	    "T_FECHO_EV4.1_HMI".TON(IN := NOT "EV4.1",                  //Quando EV4.1 recebe sinal para fechar, inicia uma contagem
	                            PT := "Inputs_HMI".T_POS_EVS);
	                                                                //No final da contagem avalia se a EV está na posição pretendida
	                                                                
	    IF ("T_ABERTURA_EV4.1_HMI".Q AND (NOT "EV4.1_ABERTA" OR ("EV4.1_ABERTA" AND "EV4.1_FECHADA"))) OR   //Condição de avaria
	        ("T_FECHO_EV4.1_HMI".Q AND (NOT "EV4.1_FECHADA" OR ("EV4.1_ABERTA" AND "EV4.1_FECHADA"))) THEN
	        #"avaria_ev4.1" := TRUE;
	    ELSE
	        #"avaria_ev4.1" := FALSE;
	    END_IF;
	                                                                
	    IF #"avaria_ev4.1" = FALSE AND "EV4.1_ABERTA" AND NOT "EV4.1_FECHADA" THEN //Condição de EV4.1 ABERTA
	        "Estados_HMI"."EV4.1_ESTADO" := 1;
	        "Estados_HMI"."EV4.1_ESTADO_PAGCMD" := 1;
	    END_IF;
	    
	    
	    IF #"avaria_ev4.1" = FALSE AND "EV4.1_FECHADA" AND NOT "EV4.1_ABERTA" THEN //Condição de EV4.1 Fechada
	        "Estados_HMI"."EV4.1_ESTADO" := 0;
	        "Estados_HMI"."EV4.1_ESTADO_PAGCMD" := 0;
	    END_IF;
	    
	    
	    IF ("T_ABERTURA_EV4.1_HMI".Q AND (NOT "EV4.1_ABERTA" OR ("EV4.1_ABERTA" AND "EV4.1_FECHADA"))) OR   //Condição de avaria
	        ("T_FECHO_EV4.1_HMI".Q AND (NOT "EV4.1_FECHADA" OR ("EV4.1_ABERTA" AND "EV4.1_FECHADA"))) THEN
	        
	        "Estados_HMI"."EV4.1_ESTADO_PAGCMD" := 2;
	        
	        CASE #"temp_clock_0.625Hz" OF
	            0:
	                "Estados_HMI"."EV4.1_ESTADO" := 0;
	            1:
	                "Estados_HMI"."EV4.1_ESTADO" := 2;
	        END_CASE;
	    END_IF;
	    
	    IF "T_ABERTURA_EV4.1_HMI".Q = FALSE AND "T_FECHO_EV4.1_HMI".Q = FALSE AND
	        "EV4.1_ABERTA" = FALSE AND "EV4.1_FECHADA" = FALSE THEN  //Condição de transição das EVs
	        
	        "Estados_HMI"."EV4.1_ESTADO_PAGCMD" := 3;
	        
	        CASE #"temp_clock_0.625Hz" OF
	            0:
	                "Estados_HMI"."EV4.1_ESTADO" := 0;
	            1:
	                "Estados_HMI"."EV4.1_ESTADO" := 3;
	        END_CASE;
	    END_IF;
	    
	END_REGION
	
	REGION Estado_EV5.1
	    
	    "T_ABERTURA_EV5.1_HMI".TON(IN := "EV5.1",                   //Quando EV5.1 recebe sinal para abrir, inicia uma contagem
	                               PT := "Inputs_HMI".T_POS_EVS);
	    
	    "T_FECHO_EV5.1_HMI".TON(IN := NOT "EV5.1",                  //Quando EV5.1 recebe sinal para fechar, inicia uma contagem
	                            PT := "Inputs_HMI".T_POS_EVS);
	                                                                //No final da contagem avalia se a EV está na posição pretendida
	                                                                
	    IF ("T_ABERTURA_EV5.1_HMI".Q AND (NOT "EV5.1_ABERTA" OR ("EV5.1_ABERTA" AND "EV5.1_FECHADA"))) OR   //Condição de avaria
	        ("T_FECHO_EV5.1_HMI".Q AND (NOT "EV5.1_FECHADA" OR ("EV5.1_ABERTA" AND "EV5.1_FECHADA"))) THEN
	        #"avaria_ev5.1" := TRUE;
	    ELSE
	        #"avaria_ev5.1" := FALSE;
	    END_IF;
	                                                                
	    IF #"avaria_ev5.1" = FALSE AND "EV5.1_ABERTA" AND NOT "EV5.1_FECHADA" THEN //Condição de EV5.1 ABERTA
	        "Estados_HMI"."EV5.1_ESTADO" := 1;
	        "Estados_HMI"."EV5.1_ESTADO_PAGCMD" := 1;
	    END_IF;
	    
	    
	    IF #"avaria_ev5.1" = FALSE AND "EV5.1_FECHADA" AND NOT "EV5.1_ABERTA" THEN //Condição de EV5.1 Fechada
	        "Estados_HMI"."EV5.1_ESTADO" := 0;
	        "Estados_HMI"."EV5.1_ESTADO_PAGCMD" := 0;
	    END_IF;
	    
	    
	    IF ("T_ABERTURA_EV5.1_HMI".Q AND (NOT "EV5.1_ABERTA" OR ("EV5.1_ABERTA" AND "EV5.1_FECHADA"))) OR   //Condição de avaria
	        ("T_FECHO_EV5.1_HMI".Q AND (NOT "EV5.1_FECHADA" OR ("EV5.1_ABERTA" AND "EV5.1_FECHADA"))) THEN
	        
	        "Estados_HMI"."EV5.1_ESTADO_PAGCMD" := 2;
	        
	        CASE #"temp_clock_0.625Hz" OF
	            0:
	                "Estados_HMI"."EV5.1_ESTADO" := 0;
	            1:
	                "Estados_HMI"."EV5.1_ESTADO" := 2;
	        END_CASE;
	    END_IF;
	    
	    IF "T_ABERTURA_EV5.1_HMI".Q = FALSE AND "T_FECHO_EV5.1_HMI".Q = FALSE AND
	        "EV5.1_ABERTA" = FALSE AND "EV5.1_FECHADA" = FALSE THEN  //Condição de transição das EVs
	        
	        "Estados_HMI"."EV5.1_ESTADO_PAGCMD" := 3;
	        
	        CASE #"temp_clock_0.625Hz" OF
	            0:
	                "Estados_HMI"."EV5.1_ESTADO" := 0;
	            1:
	                "Estados_HMI"."EV5.1_ESTADO" := 3;
	        END_CASE;
	    END_IF;
	    
	END_REGION
	
	//FILTRO 2
	
	REGION Estado_EV1.2
	    "T_ABERTURA_EV1.2_HMI".TON(IN := "EV1.2",                   //Quando EV1.2 recebe sinal para abrir, inicia uma contagem
	                               PT := "Inputs_HMI".T_POS_EVS);
	    
	    "T_FECHO_EV1.2_HMI".TON(IN := NOT "EV1.2",                  //Quando EV1.2 recebe sinal para fechar, inicia uma contagem
	                            PT := "Inputs_HMI".T_POS_EVS);
	    //No final da contagem avalia se a EV está na posição pretendida
	    
	    IF ("T_ABERTURA_EV1.2_HMI".Q AND (NOT "EV1.2_ABERTA" OR ("EV1.2_ABERTA" AND "EV1.2_FECHADA"))) OR   //Condição de avaria
	        ("T_FECHO_EV1.2_HMI".Q AND (NOT "EV1.2_FECHADA" OR ("EV1.2_ABERTA" AND "EV1.2_FECHADA"))) THEN
	        #"avaria_ev1.2" := TRUE;
	    ELSE
	        #"avaria_ev1.2" := FALSE;
	    END_IF;
	        
	    IF #"avaria_ev1.2" = FALSE AND "EV1.2_ABERTA" AND NOT "EV1.2_FECHADA" THEN //Condição de EV1.2 ABERTA
	        "Estados_HMI"."EV1.2_ESTADO" := 1;
	        "Estados_HMI"."EV1.2_ESTADO_PAGCMD" := 1;
	    END_IF;
	    
	    
	    IF #"avaria_ev1.2" = FALSE AND "EV1.2_FECHADA" AND NOT "EV1.2_ABERTA" THEN //Condição de EV1.2 Fechada
	        "Estados_HMI"."EV1.2_ESTADO" := 0;
	        "Estados_HMI"."EV1.2_ESTADO_PAGCMD" := 0;
	    END_IF;
	    
	    
	    IF ("T_ABERTURA_EV1.2_HMI".Q AND (NOT "EV1.2_ABERTA" OR ("EV1.2_ABERTA" AND "EV1.2_FECHADA"))) OR   //Condição de avaria
	        ("T_FECHO_EV1.2_HMI".Q AND (NOT "EV1.2_FECHADA" OR ("EV1.2_ABERTA" AND "EV1.2_FECHADA"))) THEN
	        
	        "Estados_HMI"."EV1.2_ESTADO_PAGCMD" := 2;
	        
	        CASE #"temp_clock_0.625Hz" OF
	            0:
	                "Estados_HMI"."EV1.2_ESTADO" := 0;
	            1:
	                "Estados_HMI"."EV1.2_ESTADO" := 2;
	        END_CASE;
	    END_IF;
	    
	    IF "T_ABERTURA_EV1.2_HMI".Q = FALSE AND "T_FECHO_EV1.2_HMI".Q = FALSE AND
	        "EV1.2_ABERTA" = FALSE AND "EV1.2_FECHADA" = FALSE THEN  //Condição de transição das EVs
	        
	        "Estados_HMI"."EV1.2_ESTADO_PAGCMD" := 3;
	        
	        CASE #"temp_clock_0.625Hz" OF
	            0:
	                "Estados_HMI"."EV1.2_ESTADO" := 0;
	            1:
	                "Estados_HMI"."EV1.2_ESTADO" := 3;
	        END_CASE;
	    END_IF;
	    
	END_REGION
	
	REGION Estado_EV2.2
	    
	    "T_ABERTURA_EV2.2_HMI".TON(IN := "EV2.2",                   //Quando EV2.2 recebe sinal para abrir, inicia uma contagem
	                               PT := "Inputs_HMI".T_POS_EVS);
	    
	    "T_FECHO_EV2.2_HMI".TON(IN := NOT "EV2.2",                  //Quando EV2.2 recebe sinal para fechar, inicia uma contagem
	                            PT := "Inputs_HMI".T_POS_EVS);
	    //No final da contagem avalia se a EV está na posição pretendida
	    
	    IF ("T_ABERTURA_EV2.2_HMI".Q AND (NOT "EV2.2_ABERTA" OR ("EV2.2_ABERTA" AND "EV2.2_FECHADA"))) OR   //Condição de avaria
	        ("T_FECHO_EV2.2_HMI".Q AND (NOT "EV2.2_FECHADA" OR ("EV2.2_ABERTA" AND "EV2.2_FECHADA"))) THEN
	        #"avaria_ev2.2" := TRUE;
	    ELSE
	        #"avaria_ev2.2" := FALSE;
	    END_IF;
	    
	    IF #"avaria_ev2.2" = FALSE AND "EV2.2_ABERTA" AND NOT "EV2.2_FECHADA" THEN //Condição de EV2.2 ABERTA
	        "Estados_HMI"."EV2.2_ESTADO" := 1;
	        "Estados_HMI"."EV2.2_ESTADO_PAGCMD" := 1;
	    END_IF;
	    
	    
	    IF #"avaria_ev2.2" = FALSE AND "EV2.2_FECHADA" AND NOT "EV2.2_ABERTA" THEN //Condição de EV2.2 Fechada
	        "Estados_HMI"."EV2.2_ESTADO" := 0;
	        "Estados_HMI"."EV2.2_ESTADO_PAGCMD" := 0;
	    END_IF;
	    
	    
	    IF ("T_ABERTURA_EV2.2_HMI".Q AND (NOT "EV2.2_ABERTA" OR ("EV2.2_ABERTA" AND "EV2.2_FECHADA"))) OR   //Condição de avaria
	        ("T_FECHO_EV2.2_HMI".Q AND (NOT "EV2.2_FECHADA" OR ("EV2.2_ABERTA" AND "EV2.2_FECHADA"))) THEN
	        
	        "Estados_HMI"."EV2.2_ESTADO_PAGCMD" := 2;
	        
	        CASE #"temp_clock_0.625Hz" OF
	            0:
	                "Estados_HMI"."EV2.2_ESTADO" := 0;
	            1:
	                "Estados_HMI"."EV2.2_ESTADO" := 2;
	        END_CASE;
	    END_IF;
	    
	    IF "T_ABERTURA_EV2.2_HMI".Q = FALSE AND "T_FECHO_EV2.2_HMI".Q = FALSE AND
	        "EV2.2_ABERTA" = FALSE AND "EV2.2_FECHADA" = FALSE THEN  //Condição de transição das EVs
	        
	        "Estados_HMI"."EV2.2_ESTADO_PAGCMD" := 3;
	        
	        CASE #"temp_clock_0.625Hz" OF
	            0:
	                "Estados_HMI"."EV2.2_ESTADO" := 0;
	            1:
	                "Estados_HMI"."EV2.2_ESTADO" := 3;
	        END_CASE;
	    END_IF;
	    
	END_REGION
	
	REGION Estado_EV3.2
	    
	    "T_ABERTURA_EV3.2_HMI".TON(IN := "EV3.2",                   //Quando EV3.2 recebe sinal para abrir, inicia uma contagem
	                               PT := "Inputs_HMI".T_POS_EVS);
	    
	    "T_FECHO_EV3.2_HMI".TON(IN := NOT "EV3.2",                  //Quando EV3.2 recebe sinal para fechar, inicia uma contagem
	                            PT := "Inputs_HMI".T_POS_EVS);
	    //No final da contagem avalia se a EV está na posição pretendida
	    
	    IF ("T_ABERTURA_EV3.2_HMI".Q AND (NOT "EV3.2_ABERTA" OR ("EV3.2_ABERTA" AND "EV3.2_FECHADA"))) OR   //Condição de avaria
	        ("T_FECHO_EV3.2_HMI".Q AND (NOT "EV3.2_FECHADA" OR ("EV3.2_ABERTA" AND "EV3.2_FECHADA"))) THEN
	        #"avaria_ev3.2" := TRUE;
	    ELSE
	        #"avaria_ev3.2" := FALSE;
	    END_IF;
	        
	    
	    IF #"avaria_ev3.2" = FALSE AND "EV3.2_ABERTA" AND NOT "EV3.2_FECHADA" THEN //Condição de EV3.2 ABERTA
	        "Estados_HMI"."EV3.2_ESTADO" := 1;
	        "Estados_HMI"."EV3.2_ESTADO_PAGCMD" := 1;
	    END_IF;
	    
	    
	    IF #"avaria_ev3.2" = FALSE AND "EV3.2_FECHADA" AND NOT "EV3.2_ABERTA" THEN //Condição de EV3.2 Fechada
	        "Estados_HMI"."EV3.2_ESTADO" := 0;
	        "Estados_HMI"."EV3.2_ESTADO_PAGCMD" := 0;
	    END_IF;
	    
	    
	    IF ("T_ABERTURA_EV3.2_HMI".Q AND (NOT "EV3.2_ABERTA" OR ("EV3.2_ABERTA" AND "EV3.2_FECHADA"))) OR   //Condição de avaria
	        ("T_FECHO_EV3.2_HMI".Q AND (NOT "EV3.2_FECHADA" OR ("EV3.2_ABERTA" AND "EV3.2_FECHADA"))) THEN
	        
	        "Estados_HMI"."EV3.2_ESTADO_PAGCMD" := 2;
	        
	        CASE #"temp_clock_0.625Hz" OF
	            0:
	                "Estados_HMI"."EV3.2_ESTADO" := 0;
	            1:
	                "Estados_HMI"."EV3.2_ESTADO" := 2;
	        END_CASE;
	    END_IF;
	    
	    IF "T_ABERTURA_EV3.2_HMI".Q = FALSE AND "T_FECHO_EV3.2_HMI".Q = FALSE AND
	        "EV3.2_ABERTA" = FALSE AND "EV3.2_FECHADA" = FALSE THEN  //Condição de transição das EVs
	        
	        "Estados_HMI"."EV3.2_ESTADO_PAGCMD" := 3;
	        
	        CASE #"temp_clock_0.625Hz" OF
	            0:
	                "Estados_HMI"."EV3.2_ESTADO" := 0;
	            1:
	                "Estados_HMI"."EV3.2_ESTADO" := 3;
	        END_CASE;
	    END_IF;
	    
	END_REGION
	
	REGION Estado_EV4.2
	    
	    "T_ABERTURA_EV4.2_HMI".TON(IN := "EV4.2",                   //Quando EV4.2 recebe sinal para abrir, inicia uma contagem
	                               PT := "Inputs_HMI".T_POS_EVS);
	    
	    "T_FECHO_EV4.2_HMI".TON(IN := NOT "EV4.2",                  //Quando EV4.2 recebe sinal para fechar, inicia uma contagem
	                            PT := "Inputs_HMI".T_POS_EVS);
	    //No final da contagem avalia se a EV está na posição pretendida
	    
	    IF ("T_ABERTURA_EV4.2_HMI".Q AND (NOT "EV4.2_ABERTA" OR ("EV4.2_ABERTA" AND "EV4.2_FECHADA"))) OR   //Condição de avaria
	        ("T_FECHO_EV4.2_HMI".Q AND (NOT "EV4.2_FECHADA" OR ("EV4.2_ABERTA" AND "EV4.2_FECHADA"))) THEN
	        #"avaria_ev4.2" := TRUE;
	    ELSE
	        #"avaria_ev4.2" := FALSE;
	    END_IF;
	    
	    
	    IF #"avaria_ev4.2" = FALSE AND "EV4.2_ABERTA" AND NOT "EV4.2_FECHADA" THEN //Condição de EV4.2 ABERTA
	        "Estados_HMI"."EV4.2_ESTADO" := 1;
	        "Estados_HMI"."EV4.2_ESTADO_PAGCMD" := 1;
	    END_IF;
	    
	    
	    IF #"avaria_ev4.2" = FALSE AND "EV4.2_FECHADA" AND NOT "EV4.2_ABERTA" THEN //Condição de EV4.2 Fechada
	        "Estados_HMI"."EV4.2_ESTADO" := 0;
	        "Estados_HMI"."EV4.2_ESTADO_PAGCMD" := 0;
	    END_IF;
	    
	    
	    IF ("T_ABERTURA_EV4.2_HMI".Q AND (NOT "EV4.2_ABERTA" OR ("EV4.2_ABERTA" AND "EV4.2_FECHADA"))) OR   //Condição de avaria
	        ("T_FECHO_EV4.2_HMI".Q AND (NOT "EV4.2_FECHADA" OR ("EV4.2_ABERTA" AND "EV4.2_FECHADA"))) THEN
	        
	        "Estados_HMI"."EV4.2_ESTADO_PAGCMD" := 2;
	        
	        CASE #"temp_clock_0.625Hz" OF
	            0:
	                "Estados_HMI"."EV4.2_ESTADO" := 0;
	            1:
	                "Estados_HMI"."EV4.2_ESTADO" := 2;
	        END_CASE;
	    END_IF;
	    
	    IF "T_ABERTURA_EV4.2_HMI".Q = FALSE AND "T_FECHO_EV4.2_HMI".Q = FALSE AND
	        "EV4.2_ABERTA" = FALSE AND "EV4.2_FECHADA" = FALSE THEN  //Condição de transição das EVs
	        
	        "Estados_HMI"."EV4.2_ESTADO_PAGCMD" := 3;
	        
	        CASE #"temp_clock_0.625Hz" OF
	            0:
	                "Estados_HMI"."EV4.2_ESTADO" := 0;
	            1:
	                "Estados_HMI"."EV4.2_ESTADO" := 3;
	        END_CASE;
	    END_IF;
	    
	END_REGION
	
	REGION Estado_EV5.2
	    
	    "T_ABERTURA_EV5.2_HMI".TON(IN := "EV5.2",                   //Quando EV5.2 recebe sinal para abrir, inicia uma contagem
	                               PT := "Inputs_HMI".T_POS_EVS);
	    
	    "T_FECHO_EV5.2_HMI".TON(IN := NOT "EV5.2",                  //Quando EV5.2 recebe sinal para fechar, inicia uma contagem
	                            PT := "Inputs_HMI".T_POS_EVS);
	    //No final da contagem avalia se a EV está na posição pretendida
	    
	    IF ("T_ABERTURA_EV5.2_HMI".Q AND (NOT "EV5.2_ABERTA" OR ("EV5.2_ABERTA" AND "EV5.2_FECHADA"))) OR   //Condição de avaria
	        ("T_FECHO_EV5.2_HMI".Q AND (NOT "EV5.2_FECHADA" OR ("EV5.2_ABERTA" AND "EV5.2_FECHADA"))) THEN
	        #"avaria_ev5.2" := TRUE;
	    ELSE
	        #"avaria_ev5.2" := FALSE;
	    END_IF;
	    
	    
	    IF #"avaria_ev5.2" = FALSE AND "EV5.2_ABERTA" AND NOT "EV5.2_FECHADA" THEN //Condição de EV5.2 ABERTA
	        "Estados_HMI"."EV5.2_ESTADO" := 1;
	        "Estados_HMI"."EV5.2_ESTADO_PAGCMD" := 1;
	    END_IF;
	    
	    
	    IF #"avaria_ev5.2" = FALSE AND "EV5.2_FECHADA" AND NOT "EV5.2_ABERTA" THEN //Condição de EV5.2 Fechada
	        "Estados_HMI"."EV5.2_ESTADO" := 0;
	        "Estados_HMI"."EV5.2_ESTADO_PAGCMD" := 0;
	    END_IF;
	    
	    
	    IF ("T_ABERTURA_EV5.2_HMI".Q AND (NOT "EV5.2_ABERTA" OR ("EV5.2_ABERTA" AND "EV5.2_FECHADA"))) OR   //Condição de avaria
	        ("T_FECHO_EV5.2_HMI".Q AND (NOT "EV5.2_FECHADA" OR ("EV5.2_ABERTA" AND "EV5.2_FECHADA"))) THEN
	        
	        "Estados_HMI"."EV5.2_ESTADO_PAGCMD" := 2;
	        
	        CASE #"temp_clock_0.625Hz" OF
	            0:
	                "Estados_HMI"."EV5.2_ESTADO" := 0;
	            1:
	                "Estados_HMI"."EV5.2_ESTADO" := 2;
	        END_CASE;
	    END_IF;
	    
	    IF "T_ABERTURA_EV5.2_HMI".Q = FALSE AND "T_FECHO_EV5.2_HMI".Q = FALSE AND
	        "EV5.2_ABERTA" = FALSE AND "EV5.2_FECHADA" = FALSE THEN  //Condição de transição das EVs
	        
	        "Estados_HMI"."EV5.2_ESTADO_PAGCMD" := 3;
	        
	        CASE #"temp_clock_0.625Hz" OF
	            0:
	                "Estados_HMI"."EV5.2_ESTADO" := 0;
	            1:
	                "Estados_HMI"."EV5.2_ESTADO" := 3;
	        END_CASE;
	    END_IF;
	    
	END_REGION
END_FUNCTION

FUNCTION "Controlo_Pressostatos" : Void   // FC8, LAD
TITLE = Ao fim de 30s indica que atingiu setpoint de pressão
{ S7_Optimized_Access := 'TRUE' }
VERSION : 0.1
// stored: AutoNumber true, IsIECCheckEnabled false, SetENOAutomatically false, UDAEnableTagReadback false
BEGIN

REGION Network 1: Pressostato Filtro 1
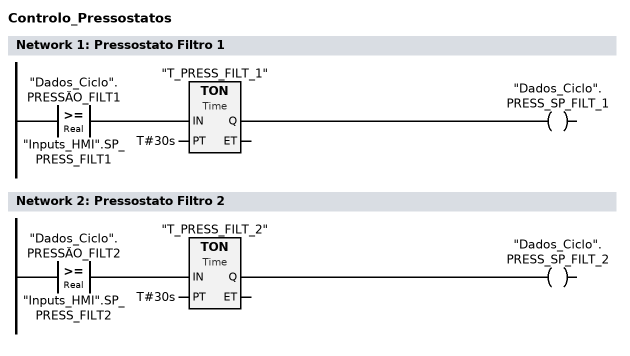
   RUNG wire#powerrail
      { S7_Templates := "SrcType := Real" } GE_Contact(in1 := "Dados_Ciclo".PRESSÃO_FILT1, in2 := "Inputs_HMI".SP_PRESS_FILT1)
      { S7_Templates := "time_type := Time" } "T_PRESS_FILT_1".TON(pt := T#30s, et =>)
      Coil( "Dados_Ciclo".PRESS_SP_FILT_1 )
   END_RUNG
   // the same network as SCL:
   "T_PRESS_FILT_1".TON(IN := "Dados_Ciclo".PRESSÃO_FILT1 >= "Inputs_HMI".SP_PRESS_FILT1, PT := T#30s);
   "Dados_Ciclo".PRESS_SP_FILT_1 := "T_PRESS_FILT_1".Q;
END_REGION

REGION Network 2: Pressostato Filtro 2
   RUNG wire#powerrail
      { S7_Templates := "SrcType := Real" } GE_Contact(in1 := "Dados_Ciclo".PRESSÃO_FILT2, in2 := "Inputs_HMI".SP_PRESS_FILT2)
      { S7_Templates := "time_type := Time" } "T_PRESS_FILT_2".TON(pt := T#30s, et =>)
      Coil( "Dados_Ciclo".PRESS_SP_FILT_2 )
   END_RUNG
   // the same network as SCL:
   "T_PRESS_FILT_2".TON(IN := "Dados_Ciclo".PRESSÃO_FILT2 >= "Inputs_HMI".SP_PRESS_FILT2, PT := T#30s);
   "Dados_Ciclo".PRESS_SP_FILT_2 := "T_PRESS_FILT_2".Q;
END_REGION
END_FUNCTION

FUNCTION "T_Func_Bombas" : Void   // FC9, LAD
{ S7_Optimized_Access := 'TRUE' }
VERSION : 0.1
// stored: AutoNumber true, IsIECCheckEnabled false, SetENOAutomatically false, UDAEnableTagReadback false
   VAR_TEMP   // added for the SCL form of the ladder/FBD networks
      _w1 : Bool;
   END_VAR
BEGIN

REGION Network 1: Período de tempo de alternancia das bombas
   // Se contador = 0, trabalha B1 e B2. Se = 1, trabalha B1 e B3. Se = 2, trabalha B2 e B3
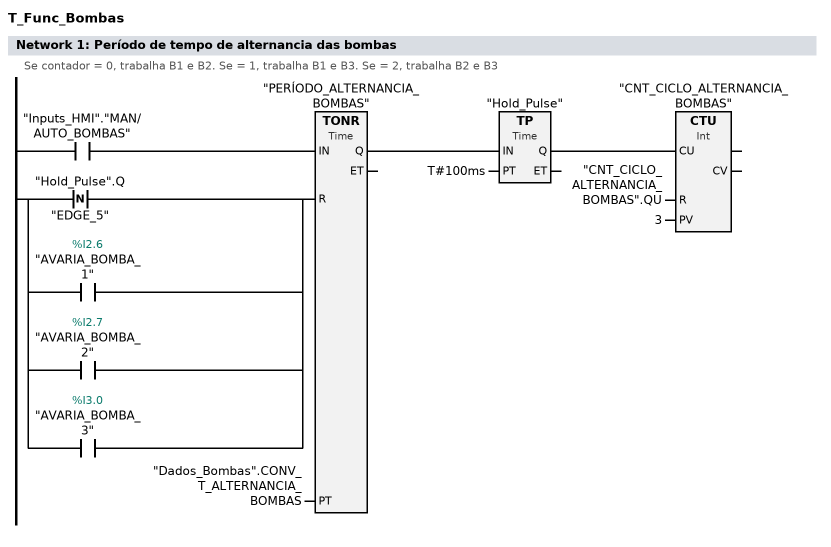
   RUNG wire#powerrail
      Contact( "Inputs_HMI"."MAN/AUTO_BOMBAS" )
      { S7_Templates := "time_type := Time" } "PERÍODO_ALTERNANCIA_BOMBAS".TONR(r := wire#w1, pt := "Dados_Bombas".CONV_T_ALTERNANCIA_BOMBAS, et =>)
      { S7_Templates := "time_type := Time" } "Hold_Pulse".TP(pt := T#100ms, et =>)
      { S7_Templates := "value_type := Int" } "CNT_CICLO_ALTERNANCIA_BOMBAS".CTU(r := "CNT_CICLO_ALTERNANCIA_BOMBAS".QU, pv := 3, cv =>)
   END_RUNG
   RUNG wire#powerrail
      N_Contact(operand := "Hold_Pulse".Q, bit := "EDGE_5")
   END_RUNG wire#w1
   RUNG wire#powerrail
      Contact( "AVARIA_BOMBA_1" )
   END_RUNG wire#w1
   RUNG wire#powerrail
      Contact( "AVARIA_BOMBA_2" )
   END_RUNG wire#w1
   RUNG wire#powerrail
      Contact( "AVARIA_BOMBA_3" )
   END_RUNG wire#w1
   // the same network as SCL:
   #_w1 := NOT "Hold_Pulse".Q AND "EDGE_5";   // falling edge of "Hold_Pulse".Q
   "EDGE_5" := "Hold_Pulse".Q;
   "PERÍODO_ALTERNANCIA_BOMBAS".TONR(IN := "Inputs_HMI"."MAN/AUTO_BOMBAS",
                           R := #_w1 OR "AVARIA_BOMBA_1" OR "AVARIA_BOMBA_2" OR "AVARIA_BOMBA_3",
                           PT := "Dados_Bombas".CONV_T_ALTERNANCIA_BOMBAS);
   "Hold_Pulse".TP(IN := "PERÍODO_ALTERNANCIA_BOMBAS".Q, PT := T#100ms);
   "CNT_CICLO_ALTERNANCIA_BOMBAS".CTU(CU := "Hold_Pulse".Q, R := "CNT_CICLO_ALTERNANCIA_BOMBAS".QU, PV := 3);
END_REGION
END_FUNCTION

FUNCTION "Conversão_Tempo_Bombas" : Void
{ S7_Optimized_Access := 'TRUE' }
VERSION : 0.1
   VAR_TEMP 
      decimal_b2 : Real;
      result_b2 : Real;
      decimal_b3 : Real;
      result_b3 : Real;
      decimal_TON : Real;
      decimal_TOFF : Real;
      result_TON : Real;
      result_TOFF : Real;
   END_VAR


BEGIN
	//Conversão do tempo de alternancia das bombas introduzido na hmi (ex: em vez de introduzir 1.5 para dar 1h30m,
	//introduz-se 1.3 para da 1h30m
	
	
	//conversão T_ALTERNANCIA bombas 
	//
	#decimal_TON := ("Inputs_HMI".T_ALTERNANCIA_BOMBAS - TRUNC("Inputs_HMI".T_ALTERNANCIA_BOMBAS)) * 1.6667;
	#result_TON := TRUNC("Inputs_HMI".T_ALTERNANCIA_BOMBAS) + #decimal_TON;
	
	"Dados_Bombas".CONV_T_ALTERNANCIA_BOMBAS :=
	DINT_TO_TIME(
	             REAL_TO_DINT(#result_TON * 3600000));
	
	
	REGION leitura_tempos_func_bombas_para_hmi
	    
	    
	    "Dados_Bombas".HORAS_TON_B1 := "CNT_FUNC_B1".CV;
	    
	    "Dados_Bombas".HORAS_TON_B2 := "CNT_FUNC_B2".CV;
	    
	    "Dados_Bombas".HORAS_TON_B3 := "CNT_FUNC_B3".CV;
	   
	END_REGION
	
END_FUNCTION

FUNCTION "Encrav_Inputs_HMI" : Void
{ S7_Optimized_Access := 'TRUE' }
VERSION : 0.1

BEGIN
	IF "Inputs_HMI"."MAN/AUTO_BOMBAS" = TRUE THEN
	    
	    "Inputs_HMI".ON_OFF_BOMBA_1 := FALSE;
	    "Inputs_HMI".ON_OFF_BOMBA_2 := FALSE;
	    "Inputs_HMI".ON_OFF_BOMBA_3 := FALSE;
	    
	END_IF;
	
	IF "Inputs_HMI"."MAN/AUTO" = TRUE THEN
	    
	    "Inputs_HMI"."ON_OFF_EV1.1" := FALSE;
	    "Inputs_HMI"."ON_OFF_EV2.1" := FALSE;
	    "Inputs_HMI"."ON_OFF_EV3.1" := FALSE;
	    "Inputs_HMI"."ON_OFF_EV4.1" := FALSE;
	    "Inputs_HMI"."ON_OFF_EV5.1" := FALSE;
	    
	    "Inputs_HMI"."ON_OFF_EV1.2" := FALSE;
	    "Inputs_HMI"."ON_OFF_EV2.2" := FALSE;
	    "Inputs_HMI"."ON_OFF_EV3.2" := FALSE;
	    "Inputs_HMI"."ON_OFF_EV4.2" := FALSE;
	    "Inputs_HMI"."ON_OFF_EV5.2" := FALSE;
	 
	END_IF;
	
END_FUNCTION

FUNCTION "Conversão_TLAV_TRINSE" : Void
{ S7_Optimized_Access := 'TRUE' }
VERSION : 0.1

BEGIN
	//Conversão do tempo decorrido de lavagem e enxaguamento para minutos
	
	"Estados_HMI".T_LAV_MINUTOS := (TIME_TO_DINT("T_LAVAGEM".ET) MOD 3600000) / 60000;
	"Estados_HMI".T_RINSE_MINUTOS := (TIME_TO_DINT("T_RINSE".ET) MOD 3600000) / 60000;
END_FUNCTION

FUNCTION "Alarmes" : Void
{ S7_Optimized_Access := 'TRUE' }
VERSION : 0.1

BEGIN
	//Alarmes filtro 1
	//
	REGION ALARME_V1.1
	    IF "T_ABERTURA_EV1.1_HMI".Q AND NOT "EV1.1_ABERTA" THEN  //Válvula não abriu
	        "Estados_HMI".ALARMES_LISTA_1.%X0 := TRUE;
	    ELSE
	        "Estados_HMI".ALARMES_LISTA_1.%X0 := FALSE;
	    END_IF;
	    
	    
	    IF "T_ABERTURA_EV1.1_HMI".Q AND "EV1.1_ABERTA" AND "EV1.1_FECHADA" THEN  //Avaria fim de curso de fecho
	        "Estados_HMI".ALARMES_LISTA_1.%X1 := TRUE;
	    ELSE
	        "Estados_HMI".ALARMES_LISTA_1.%X1 := FALSE;
	    END_IF;
	    
	    
	    IF "T_FECHO_EV1.1_HMI".Q AND NOT "EV1.1_FECHADA" THEN  //Válvula não fechou
	        "Estados_HMI".ALARMES_LISTA_1.%X2 := TRUE;
	    ELSE
	        "Estados_HMI".ALARMES_LISTA_1.%X2 := FALSE;
	    END_IF;
	    
	    
	    IF "T_FECHO_EV1.1_HMI".Q AND "EV1.1_ABERTA" AND "EV1.1_FECHADA" THEN  //Avaria fim de curso de abertura
	        "Estados_HMI".ALARMES_LISTA_1.%X3 := TRUE;
	    ELSE
	        "Estados_HMI".ALARMES_LISTA_1.%X3 := FALSE;
	    END_IF;
	END_REGION
	REGION ALARME_V2.1
	    IF "T_ABERTURA_EV2.1_HMI".Q AND NOT "EV2.1_ABERTA" THEN  //Válvula não abriu
	        "Estados_HMI".ALARMES_LISTA_1.%X4 := TRUE;
	    ELSE
	        "Estados_HMI".ALARMES_LISTA_1.%X4 := FALSE;
	    END_IF;
	    
	    
	    IF "T_ABERTURA_EV2.1_HMI".Q AND "EV2.1_ABERTA" AND "EV2.1_FECHADA" THEN  //Avaria fim de curso de fecho
	        "Estados_HMI".ALARMES_LISTA_1.%X5 := TRUE;
	    ELSE
	        "Estados_HMI".ALARMES_LISTA_1.%X5 := FALSE;
	    END_IF;
	    
	    
	    IF "T_FECHO_EV2.1_HMI".Q AND NOT "EV2.1_FECHADA" THEN  //Válvula não fechou
	        "Estados_HMI".ALARMES_LISTA_1.%X6 := TRUE;
	    ELSE
	        "Estados_HMI".ALARMES_LISTA_1.%X6 := FALSE;
	    END_IF;
	    
	    
	    IF "T_FECHO_EV2.1_HMI".Q AND "EV2.1_ABERTA" AND "EV2.1_FECHADA" THEN  //Avaria fim de curso de abertura
	        "Estados_HMI".ALARMES_LISTA_1.%X7 := TRUE;
	    ELSE
	        "Estados_HMI".ALARMES_LISTA_1.%X7 := FALSE;
	    END_IF;
	END_REGION
	REGION ALARME_V3.1
	    IF "T_ABERTURA_EV3.1_HMI".Q AND NOT "EV3.1_ABERTA" THEN  //Válvula não abriu
	        "Estados_HMI".ALARMES_LISTA_1.%X8 := TRUE;
	    ELSE
	        "Estados_HMI".ALARMES_LISTA_1.%X8 := FALSE;
	    END_IF;
	    
	    
	    IF "T_ABERTURA_EV3.1_HMI".Q AND "EV3.1_ABERTA" AND "EV3.1_FECHADA" THEN  //Avaria fim de curso de fecho
	        "Estados_HMI".ALARMES_LISTA_1.%X9 := TRUE;
	    ELSE
	        "Estados_HMI".ALARMES_LISTA_1.%X9 := FALSE;
	    END_IF;
	    
	    
	    IF "T_FECHO_EV3.1_HMI".Q AND NOT "EV3.1_FECHADA" THEN  //Válvula não fechou
	        "Estados_HMI".ALARMES_LISTA_1.%X10 := TRUE;
	    ELSE
	        "Estados_HMI".ALARMES_LISTA_1.%X10 := FALSE;
	    END_IF;
	    
	    
	    IF "T_FECHO_EV3.1_HMI".Q AND "EV3.1_ABERTA" AND "EV3.1_FECHADA" THEN  //Avaria fim de curso de abertura
	        "Estados_HMI".ALARMES_LISTA_1.%X11 := TRUE;
	    ELSE
	        "Estados_HMI".ALARMES_LISTA_1.%X11 := FALSE;
	    END_IF;
	END_REGION
	REGION ALARME_V4.1
	    IF "T_ABERTURA_EV4.1_HMI".Q AND NOT "EV4.1_ABERTA" THEN  //Válvula não abriu
	        "Estados_HMI".ALARMES_LISTA_1.%X12 := TRUE;
	    ELSE
	        "Estados_HMI".ALARMES_LISTA_1.%X12 := FALSE;
	    END_IF;
	    
	    
	    IF "T_ABERTURA_EV4.1_HMI".Q AND "EV4.1_ABERTA" AND "EV4.1_FECHADA" THEN  //Avaria fim de curso de fecho
	        "Estados_HMI".ALARMES_LISTA_1.%X13 := TRUE;
	    ELSE
	        "Estados_HMI".ALARMES_LISTA_1.%X13 := FALSE;
	    END_IF;
	    
	    
	    IF "T_FECHO_EV4.1_HMI".Q AND NOT "EV4.1_FECHADA" THEN  //Válvula não fechou
	        "Estados_HMI".ALARMES_LISTA_1.%X14 := TRUE;
	    ELSE
	        "Estados_HMI".ALARMES_LISTA_1.%X14 := FALSE;
	    END_IF;
	    
	    
	    IF "T_FECHO_EV4.1_HMI".Q AND "EV4.1_ABERTA" AND "EV4.1_FECHADA" THEN  //Avaria fim de curso de abertura
	        "Estados_HMI".ALARMES_LISTA_1.%X15 := TRUE;
	    ELSE
	        "Estados_HMI".ALARMES_LISTA_1.%X15 := FALSE;
	    END_IF;
	END_REGION
	REGION ALARME_V5.1
	    IF "T_ABERTURA_EV5.1_HMI".Q AND NOT "EV5.1_ABERTA" THEN  //Válvula não abriu
	        "Estados_HMI".ALARMES_LISTA_2.%X0 := TRUE;
	    ELSE
	        "Estados_HMI".ALARMES_LISTA_2.%X0 := FALSE;
	    END_IF;
	    
	    
	    IF "T_ABERTURA_EV5.1_HMI".Q AND "EV5.1_ABERTA" AND "EV5.1_FECHADA" THEN  //Avaria fim de curso de fecho
	        "Estados_HMI".ALARMES_LISTA_2.%X1 := TRUE;
	    ELSE
	        "Estados_HMI".ALARMES_LISTA_2.%X1 := FALSE;
	    END_IF;
	    
	    
	    IF "T_FECHO_EV5.1_HMI".Q AND NOT "EV5.1_FECHADA" THEN  //Válvula não fechou
	        "Estados_HMI".ALARMES_LISTA_2.%X2 := TRUE;
	    ELSE
	        "Estados_HMI".ALARMES_LISTA_2.%X2 := FALSE;
	    END_IF;
	    
	    
	    IF "T_FECHO_EV5.1_HMI".Q AND "EV5.1_ABERTA" AND "EV5.1_FECHADA" THEN  //Avaria fim de curso de abertura
	        "Estados_HMI".ALARMES_LISTA_2.%X3 := TRUE;
	    ELSE
	        "Estados_HMI".ALARMES_LISTA_2.%X3 := FALSE;
	    END_IF;
	END_REGION
	
	//Alarmes filtro 2
	//
	REGION ALARME_V1.2
	    IF "T_ABERTURA_EV1.2_HMI".Q AND NOT "EV1.2_ABERTA" THEN  //Válvula não abriu
	        "Estados_HMI".ALARMES_LISTA_2.%X4 := TRUE;
	    ELSE
	        "Estados_HMI".ALARMES_LISTA_2.%X4 := FALSE;
	    END_IF;
	    
	    
	    IF "T_ABERTURA_EV1.2_HMI".Q AND "EV1.2_ABERTA" AND "EV1.2_FECHADA" THEN  //Avaria fim de curso de fecho
	        "Estados_HMI".ALARMES_LISTA_2.%X5 := TRUE;
	    ELSE
	        "Estados_HMI".ALARMES_LISTA_2.%X5 := FALSE;
	    END_IF;
	    
	    
	    IF "T_FECHO_EV1.2_HMI".Q AND NOT "EV1.2_FECHADA" THEN  //Válvula não fechou
	        "Estados_HMI".ALARMES_LISTA_2.%X6 := TRUE;
	    ELSE
	        "Estados_HMI".ALARMES_LISTA_2.%X6 := FALSE;
	    END_IF;
	    
	    
	    IF "T_FECHO_EV1.2_HMI".Q AND "EV1.2_ABERTA" AND "EV1.2_FECHADA" THEN  //Avaria fim de curso de abertura
	        "Estados_HMI".ALARMES_LISTA_2.%X7 := TRUE;
	    ELSE
	        "Estados_HMI".ALARMES_LISTA_2.%X7 := FALSE;
	    END_IF;
	END_REGION
	REGION ALARME_V2.2
	    IF "T_ABERTURA_EV2.2_HMI".Q AND NOT "EV2.2_ABERTA" THEN  //Válvula não abriu
	        "Estados_HMI".ALARMES_LISTA_2.%X8 := TRUE;
	    ELSE
	        "Estados_HMI".ALARMES_LISTA_2.%X8 := FALSE;
	    END_IF;
	    
	    
	    IF "T_ABERTURA_EV2.2_HMI".Q AND "EV2.2_ABERTA" AND "EV2.2_FECHADA" THEN  //Avaria fim de curso de fecho
	        "Estados_HMI".ALARMES_LISTA_2.%X9 := TRUE;
	    ELSE
	        "Estados_HMI".ALARMES_LISTA_2.%X9 := FALSE;
	    END_IF;
	    
	    
	    IF "T_FECHO_EV2.2_HMI".Q AND NOT "EV2.2_FECHADA" THEN  //Válvula não fechou
	        "Estados_HMI".ALARMES_LISTA_2.%X10 := TRUE;
	    ELSE
	        "Estados_HMI".ALARMES_LISTA_2.%X10 := FALSE;
	    END_IF;
	    
	    
	    IF "T_FECHO_EV2.2_HMI".Q AND "EV2.2_ABERTA" AND "EV2.2_FECHADA" THEN  //Avaria fim de curso de abertura
	        "Estados_HMI".ALARMES_LISTA_2.%X11 := TRUE;
	    ELSE
	        "Estados_HMI".ALARMES_LISTA_2.%X11 := FALSE;
	    END_IF;
	END_REGION
	REGION ALARME_V3.2
	    IF "T_ABERTURA_EV3.2_HMI".Q AND NOT "EV3.2_ABERTA" THEN  //Válvula não abriu
	        "Estados_HMI".ALARMES_LISTA_2.%X12 := TRUE;
	    ELSE
	        "Estados_HMI".ALARMES_LISTA_2.%X12 := FALSE;
	    END_IF;
	    
	    
	    IF "T_ABERTURA_EV3.2_HMI".Q AND "EV3.2_ABERTA" AND "EV3.2_FECHADA" THEN  //Avaria fim de curso de fecho
	        "Estados_HMI".ALARMES_LISTA_2.%X13 := TRUE;
	    ELSE
	        "Estados_HMI".ALARMES_LISTA_2.%X13 := FALSE;
	    END_IF;
	    
	    
	    IF "T_FECHO_EV3.2_HMI".Q AND NOT "EV3.2_FECHADA" THEN  //Válvula não fechou
	        "Estados_HMI".ALARMES_LISTA_2.%X14 := TRUE;
	    ELSE
	        "Estados_HMI".ALARMES_LISTA_2.%X14 := FALSE;
	    END_IF;
	    
	    
	    IF "T_FECHO_EV3.2_HMI".Q AND "EV3.2_ABERTA" AND "EV3.2_FECHADA" THEN  //Avaria fim de curso de abertura
	        "Estados_HMI".ALARMES_LISTA_2.%X15 := TRUE;
	    ELSE
	        "Estados_HMI".ALARMES_LISTA_2.%X15 := FALSE;
	    END_IF;
	END_REGION
	REGION ALARME_V4.2
	    IF "T_ABERTURA_EV4.2_HMI".Q AND NOT "EV4.2_ABERTA" THEN  //Válvula não abriu
	        "Estados_HMI".ALARMES_LISTA_3.%X0 := TRUE;
	    ELSE
	        "Estados_HMI".ALARMES_LISTA_3.%X0 := FALSE;
	    END_IF;
	    
	    
	    IF "T_ABERTURA_EV4.2_HMI".Q AND "EV4.2_ABERTA" AND "EV4.2_FECHADA" THEN  //Avaria fim de curso de fecho
	        "Estados_HMI".ALARMES_LISTA_3.%X1 := TRUE;
	    ELSE
	        "Estados_HMI".ALARMES_LISTA_3.%X1 := FALSE;
	    END_IF;
	    
	    
	    IF "T_FECHO_EV4.2_HMI".Q AND NOT "EV4.2_FECHADA" THEN  //Válvula não fechou
	        "Estados_HMI".ALARMES_LISTA_3.%X2 := TRUE;
	    ELSE
	        "Estados_HMI".ALARMES_LISTA_3.%X2 := FALSE;
	    END_IF;
	    
	    
	    IF "T_FECHO_EV4.2_HMI".Q AND "EV4.2_ABERTA" AND "EV4.2_FECHADA" THEN  //Avaria fim de curso de abertura
	        "Estados_HMI".ALARMES_LISTA_3.%X3 := TRUE;
	    ELSE
	        "Estados_HMI".ALARMES_LISTA_3.%X3 := FALSE;
	    END_IF;
	END_REGION
	REGION ALARME_V5.2
	    IF "T_ABERTURA_EV5.2_HMI".Q AND NOT "EV5.2_ABERTA" THEN  //Válvula não abriu
	        "Estados_HMI".ALARMES_LISTA_3.%X4 := TRUE;
	    ELSE
	        "Estados_HMI".ALARMES_LISTA_3.%X4 := FALSE;
	    END_IF;
	    
	    
	    IF "T_ABERTURA_EV5.2_HMI".Q AND "EV5.2_ABERTA" AND "EV5.2_FECHADA" THEN  //Avaria fim de curso de fecho
	        "Estados_HMI".ALARMES_LISTA_3.%X5 := TRUE;
	    ELSE
	        "Estados_HMI".ALARMES_LISTA_3.%X5 := FALSE;
	    END_IF;
	    
	    
	    IF "T_FECHO_EV5.2_HMI".Q AND NOT "EV5.2_FECHADA" THEN  //Válvula não fechou
	        "Estados_HMI".ALARMES_LISTA_3.%X6 := TRUE;
	    ELSE
	        "Estados_HMI".ALARMES_LISTA_3.%X6 := FALSE;
	    END_IF;
	    
	    
	    IF "T_FECHO_EV5.2_HMI".Q AND "EV5.2_ABERTA" AND "EV5.2_FECHADA" THEN  //Avaria fim de curso de abertura
	        "Estados_HMI".ALARMES_LISTA_3.%X7 := TRUE;
	    ELSE
	        "Estados_HMI".ALARMES_LISTA_3.%X7 := FALSE;
	    END_IF;
	END_REGION
	
	//Alarmes Bombas
	//
	REGION ALARME_BOMBA_1
	    IF "AVARIA_BOMBA_1" = TRUE THEN
	        "Estados_HMI".ALARMES_LISTA_3.%X8 := TRUE;
	    ELSE
	        "Estados_HMI".ALARMES_LISTA_3.%X8 := FALSE;
	    END_IF;
	END_REGION
	
	REGION ALARME_BOMBA_2
	    IF "AVARIA_BOMBA_2" = TRUE THEN
	        "Estados_HMI".ALARMES_LISTA_3.%X9 := TRUE;
	    ELSE
	        "Estados_HMI".ALARMES_LISTA_3.%X9 := FALSE;
	    END_IF;
	END_REGION
	
	REGION ALARME_BOMBA_3
	    IF "AVARIA_BOMBA_3" = TRUE THEN
	        "Estados_HMI".ALARMES_LISTA_3.%X10 := TRUE;
	    ELSE
	        "Estados_HMI".ALARMES_LISTA_3.%X10 := FALSE;
	    END_IF;
	END_REGION
	
	
	
	
	
	
END_FUNCTION

FUNCTION "UV" : Void   // FC15, LAD
{ S7_Optimized_Access := 'TRUE' }
VERSION : 0.1
// stored: AutoNumber true, IsIECCheckEnabled false, SetENOAutomatically false, UDAEnableTagReadback false
   VAR_TEMP
      sr_ultravioleta : Bool;
   END_VAR
BEGIN

REGION Network 1
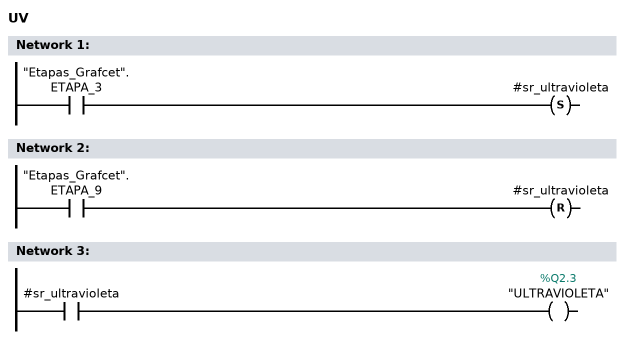
   RUNG wire#powerrail
      Contact( "Etapas_Grafcet".ETAPA_3 )
      S_Coil( #sr_ultravioleta )
   END_RUNG
   // the same network as SCL:
   IF "Etapas_Grafcet".ETAPA_3 THEN #sr_ultravioleta := TRUE; END_IF;
END_REGION

REGION Network 2
   RUNG wire#powerrail
      Contact( "Etapas_Grafcet".ETAPA_9 )
      R_Coil( #sr_ultravioleta )
   END_RUNG
   // the same network as SCL:
   IF "Etapas_Grafcet".ETAPA_9 THEN #sr_ultravioleta := FALSE; END_IF;
END_REGION

REGION Network 3
   RUNG wire#powerrail
      Contact( #sr_ultravioleta )
      Coil( "ULTRAVIOLETA" )
   END_RUNG
   // the same network as SCL:
   "ULTRAVIOLETA" := #sr_ultravioleta;
END_REGION
END_FUNCTION

FUNCTION "Ciclo_Hórario_Filtros" : Void   // FC16, LAD
{ S7_Optimized_Access := 'TRUE' }
VERSION : 0.1
// stored: AutoNumber true, IsIECCheckEnabled false, SetENOAutomatically false, UDAEnableTagReadback false
   VAR_TEMP   // added for the SCL form of the ladder/FBD networks
      _w1 : Bool;
   END_VAR
BEGIN

REGION Network 1: Leitura de tempo do sistema
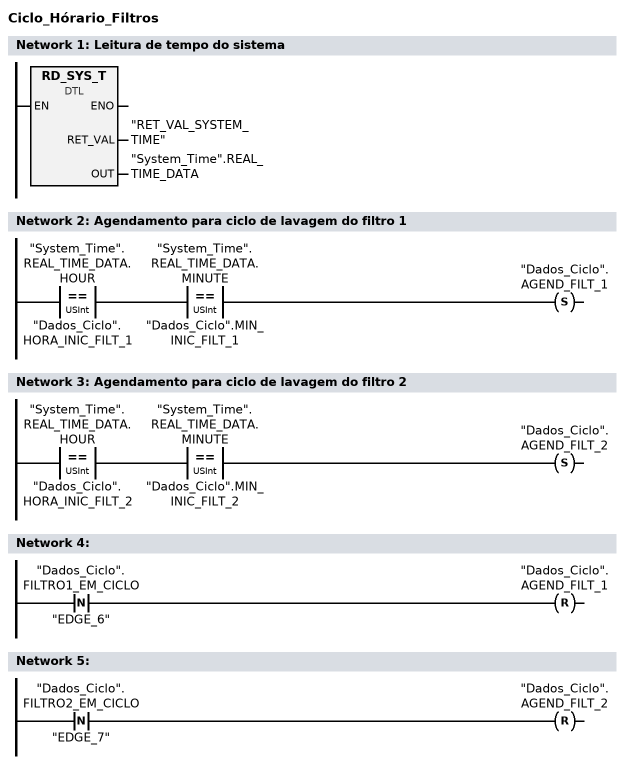
   RUNG wire#powerrail
      { S7_Templates := "date_type := DTL" } RD_SYS_T(RET_VAL => "RET_VAL_SYSTEM_TIME", OUT => "System_Time".REAL_TIME_DATA)
   END_RUNG
   // the same network as SCL:
   "RET_VAL_SYSTEM_TIME" := RD_SYS_T(OUT => "System_Time".REAL_TIME_DATA);
END_REGION

REGION Network 2: Agendamento para ciclo de lavagem do filtro 1
   RUNG wire#powerrail
      { S7_Templates := "SrcType := USInt" } EQ_Contact(in1 := "System_Time".REAL_TIME_DATA.HOUR, in2 := "Dados_Ciclo".HORA_INIC_FILT_1)
      { S7_Templates := "SrcType := USInt" } EQ_Contact(in1 := "System_Time".REAL_TIME_DATA.MINUTE, in2 := "Dados_Ciclo".MIN_INIC_FILT_1)
      S_Coil( "Dados_Ciclo".AGEND_FILT_1 )
   END_RUNG
   // the same network as SCL:
   IF ("System_Time".REAL_TIME_DATA.HOUR = "Dados_Ciclo".HORA_INIC_FILT_1) AND ("System_Time".REAL_TIME_DATA.MINUTE = "Dados_Ciclo".MIN_INIC_FILT_1) THEN
       "Dados_Ciclo".AGEND_FILT_1 := TRUE;
   END_IF;
END_REGION

REGION Network 3: Agendamento para ciclo de lavagem do filtro 2
   RUNG wire#powerrail
      { S7_Templates := "SrcType := USInt" } EQ_Contact(in1 := "System_Time".REAL_TIME_DATA.HOUR, in2 := "Dados_Ciclo".HORA_INIC_FILT_2)
      { S7_Templates := "SrcType := USInt" } EQ_Contact(in1 := "System_Time".REAL_TIME_DATA.MINUTE, in2 := "Dados_Ciclo".MIN_INIC_FILT_2)
      S_Coil( "Dados_Ciclo".AGEND_FILT_2 )
   END_RUNG
   // the same network as SCL:
   IF ("System_Time".REAL_TIME_DATA.HOUR = "Dados_Ciclo".HORA_INIC_FILT_2) AND ("System_Time".REAL_TIME_DATA.MINUTE = "Dados_Ciclo".MIN_INIC_FILT_2) THEN
       "Dados_Ciclo".AGEND_FILT_2 := TRUE;
   END_IF;
END_REGION

REGION Network 4
   RUNG wire#powerrail
      N_Contact(operand := "Dados_Ciclo".FILTRO1_EM_CICLO, bit := "EDGE_6")
      R_Coil( "Dados_Ciclo".AGEND_FILT_1 )
   END_RUNG
   // the same network as SCL:
   #_w1 := NOT "Dados_Ciclo".FILTRO1_EM_CICLO AND "EDGE_6";   // falling edge of "Dados_Ciclo".FILTRO1_EM_CICLO
   "EDGE_6" := "Dados_Ciclo".FILTRO1_EM_CICLO;
   IF #_w1 THEN "Dados_Ciclo".AGEND_FILT_1 := FALSE; END_IF;
END_REGION

REGION Network 5
   RUNG wire#powerrail
      N_Contact(operand := "Dados_Ciclo".FILTRO2_EM_CICLO, bit := "EDGE_7")
      R_Coil( "Dados_Ciclo".AGEND_FILT_2 )
   END_RUNG
   // the same network as SCL:
   #_w1 := NOT "Dados_Ciclo".FILTRO2_EM_CICLO AND "EDGE_7";   // falling edge of "Dados_Ciclo".FILTRO2_EM_CICLO
   "EDGE_7" := "Dados_Ciclo".FILTRO2_EM_CICLO;
   IF #_w1 THEN "Dados_Ciclo".AGEND_FILT_2 := FALSE; END_IF;
END_REGION
END_FUNCTION

FUNCTION "Totalizador_Bombas" : Void   // FC10, LAD
{ S7_Optimized_Access := 'TRUE' }
VERSION : 0.1
// stored: AutoNumber true, IsIECCheckEnabled false, SetENOAutomatically false, UDAEnableTagReadback false
BEGIN

REGION Network 1
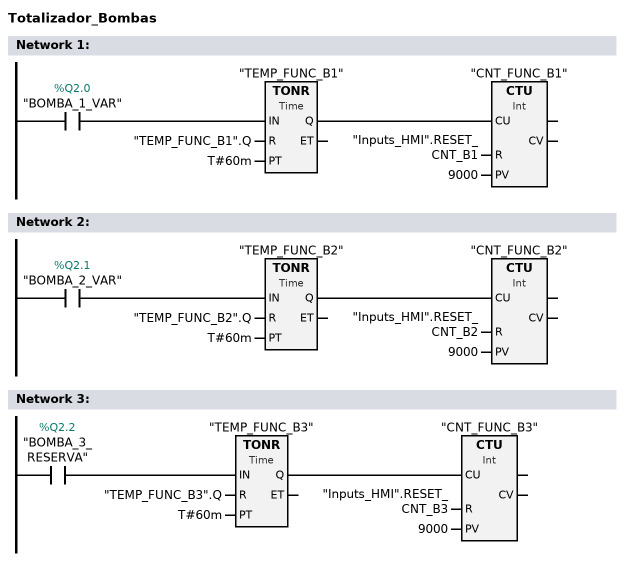
   RUNG wire#powerrail
      Contact( "BOMBA_1_VAR" )
      { S7_Templates := "time_type := Time" } "TEMP_FUNC_B1".TONR(r := "TEMP_FUNC_B1".Q, pt := T#60m, et =>)
      { S7_Templates := "value_type := Int" } "CNT_FUNC_B1".CTU(r := "Inputs_HMI".RESET_CNT_B1, pv := 9000, cv =>)
   END_RUNG
   // the same network as SCL:
   "TEMP_FUNC_B1".TONR(IN := "BOMBA_1_VAR", R := "TEMP_FUNC_B1".Q, PT := T#60m);
   "CNT_FUNC_B1".CTU(CU := "TEMP_FUNC_B1".Q, R := "Inputs_HMI".RESET_CNT_B1, PV := 9000);
END_REGION

REGION Network 2
   RUNG wire#powerrail
      Contact( "BOMBA_2_VAR" )
      { S7_Templates := "time_type := Time" } "TEMP_FUNC_B2".TONR(r := "TEMP_FUNC_B2".Q, pt := T#60m, et =>)
      { S7_Templates := "value_type := Int" } "CNT_FUNC_B2".CTU(r := "Inputs_HMI".RESET_CNT_B2, pv := 9000, cv =>)
   END_RUNG
   // the same network as SCL:
   "TEMP_FUNC_B2".TONR(IN := "BOMBA_2_VAR", R := "TEMP_FUNC_B2".Q, PT := T#60m);
   "CNT_FUNC_B2".CTU(CU := "TEMP_FUNC_B2".Q, R := "Inputs_HMI".RESET_CNT_B2, PV := 9000);
END_REGION

REGION Network 3
   RUNG wire#powerrail
      Contact( "BOMBA_3_RESERVA" )
      { S7_Templates := "time_type := Time" } "TEMP_FUNC_B3".TONR(r := "TEMP_FUNC_B3".Q, pt := T#60m, et =>)
      { S7_Templates := "value_type := Int" } "CNT_FUNC_B3".CTU(r := "Inputs_HMI".RESET_CNT_B3, pv := 9000, cv =>)
   END_RUNG
   // the same network as SCL:
   "TEMP_FUNC_B3".TONR(IN := "BOMBA_3_RESERVA", R := "TEMP_FUNC_B3".Q, PT := T#60m);
   "CNT_FUNC_B3".CTU(CU := "TEMP_FUNC_B3".Q, R := "Inputs_HMI".RESET_CNT_B3, PV := 9000);
END_REGION
END_FUNCTION

FUNCTION "Proc_Analog_Press_Filt1" : Void   // FC18, LAD
{ S7_Optimized_Access := 'TRUE' }
VERSION : 0.1
// stored: AutoNumber true, IsIECCheckEnabled false, SetENOAutomatically false, UDAEnableTagReadback false
   VAR_OUTPUT
      Pressão_em_Bar : Real;
   END_VAR
   VAR_TEMP
      "Pressão_em_%" : Real;
   END_VAR
BEGIN

REGION Network 1
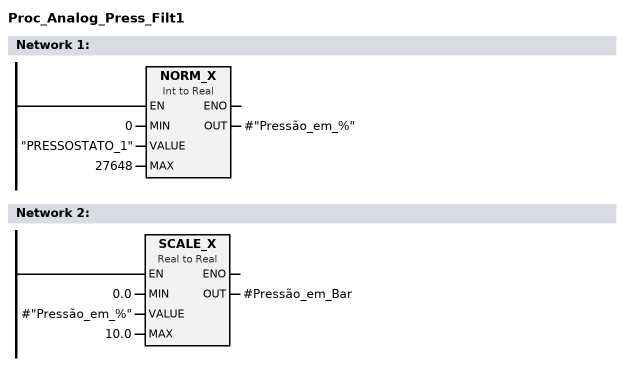
   RUNG wire#powerrail
      { S7_Templates := "[SrcType := Int, DestType := Real]"; S7_GenerateENO := "TRUE" } Normalize(min := 0, value := "PRESSOSTATO_1", max := 27648, out => #"Pressão_em_%")
   END_RUNG
   // the same network as SCL:
   #"Pressão_em_%" := NORM_X(MIN := 0, VALUE := "PRESSOSTATO_1", MAX := 27648);
END_REGION

REGION Network 2
   RUNG wire#powerrail
      { S7_Templates := "[SrcType := Real, DestType := Real]"; S7_GenerateENO := "TRUE" } Scale(min := 0.0, value := #"Pressão_em_%", max := 10.0, out => #Pressão_em_Bar)
   END_RUNG
   // the same network as SCL:
   #Pressão_em_Bar := SCALE_X(MIN := 0.0, VALUE := #"Pressão_em_%", MAX := 10.0);
END_REGION
END_FUNCTION

FUNCTION "Proc_Analog_Press_Filt2" : Void   // FC19, LAD
{ S7_Optimized_Access := 'TRUE' }
VERSION : 0.1
// stored: AutoNumber true, IsIECCheckEnabled false, SetENOAutomatically false, UDAEnableTagReadback false
   VAR_OUTPUT
      Pressão_em_Bar : Real;
   END_VAR
   VAR_TEMP
      "Pressão_em_%" : Real;
   END_VAR
BEGIN

REGION Network 1
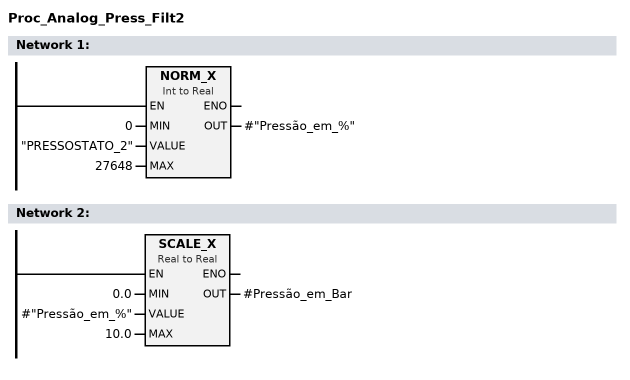
   RUNG wire#powerrail
      { S7_Templates := "[SrcType := Int, DestType := Real]"; S7_GenerateENO := "TRUE" } Normalize(min := 0, value := "PRESSOSTATO_2", max := 27648, out => #"Pressão_em_%")
   END_RUNG
   // the same network as SCL:
   #"Pressão_em_%" := NORM_X(MIN := 0, VALUE := "PRESSOSTATO_2", MAX := 27648);
END_REGION

REGION Network 2
   RUNG wire#powerrail
      { S7_Templates := "[SrcType := Real, DestType := Real]"; S7_GenerateENO := "TRUE" } Scale(min := 0.0, value := #"Pressão_em_%", max := 10.0, out => #Pressão_em_Bar)
   END_RUNG
   // the same network as SCL:
   #Pressão_em_Bar := SCALE_X(MIN := 0.0, VALUE := #"Pressão_em_%", MAX := 10.0);
END_REGION
END_FUNCTION

FUNCTION "Estado_Bombas" : Void
{ S7_Optimized_Access := 'TRUE' }
VERSION : 0.1

BEGIN
	//SINALIZAÇÃO DO ESTADO DAS BOMBAS PARA HMI
	
	REGION ESTADO_BOMBA_1
	    IF "BOMBA_1_VAR" = TRUE AND NOT "AVARIA_BOMBA_1" THEN  //BOMBA LIGADA
	        "Estados_HMI".BOMBA_1_ESTADO := 1;
	        "Estados_HMI".BOMBA_1_ESTADO_PAGCMD := 1;
	    END_IF;
	    
	    IF "BOMBA_1_VAR" = FALSE AND NOT "AVARIA_BOMBA_1" THEN  //BOMBA DESLIGADA
	        "Estados_HMI".BOMBA_1_ESTADO := 0;
	        "Estados_HMI".BOMBA_1_ESTADO_PAGCMD := 0;
	    END_IF;
	    
	    IF "AVARIA_BOMBA_1" THEN  //BOMBA AVARIA
	        "Estados_HMI".BOMBA_1_ESTADO := 2;
	        "Estados_HMI".BOMBA_1_ESTADO_PAGCMD := 2;
	    END_IF;
	END_REGION
	
	REGION ESTADO_BOMBA_2
	    IF "BOMBA_2_VAR" = TRUE AND NOT "AVARIA_BOMBA_2" THEN  //BOMBA LIGADA
	        "Estados_HMI".BOMBA_2_ESTADO := 1;
	        "Estados_HMI".BOMBA_2_ESTADO_PAGCMD := 1;
	    END_IF;
	    
	    IF "BOMBA_2_VAR" = FALSE AND NOT "AVARIA_BOMBA_2" THEN  //BOMBA DESLIGADA
	        "Estados_HMI".BOMBA_2_ESTADO := 0;
	        "Estados_HMI".BOMBA_2_ESTADO_PAGCMD := 0;
	    END_IF;
	    
	    IF "AVARIA_BOMBA_2" THEN  //BOMBA AVARIA
	        "Estados_HMI".BOMBA_2_ESTADO := 2;
	        "Estados_HMI".BOMBA_2_ESTADO_PAGCMD := 2;
	    END_IF;
	END_REGION
	
	REGION ESTADO_BOMBA_3
	    IF "BOMBA_3_RESERVA" = TRUE AND NOT "AVARIA_BOMBA_3" THEN  //BOMBA LIGADA
	        "Estados_HMI".BOMBA_3_ESTADO := 1;
	        "Estados_HMI".BOMBA_3_ESTADO_PAGCMD := 1;
	    END_IF;
	    
	    IF "BOMBA_3_RESERVA" = FALSE AND NOT "AVARIA_BOMBA_3" THEN  //BOMBA DESLIGADA
	        "Estados_HMI".BOMBA_3_ESTADO := 0;
	        "Estados_HMI".BOMBA_3_ESTADO_PAGCMD := 0;
	    END_IF;
	    
	    IF "AVARIA_BOMBA_3" THEN  //BOMBA AVARIA
	        "Estados_HMI".BOMBA_3_ESTADO := 2;
	        "Estados_HMI".BOMBA_3_ESTADO_PAGCMD := 2;
	    END_IF;
	END_REGION
END_FUNCTION

FUNCTION "Comando_Avaria_Bombas" : Void   // FC21, LAD
{ S7_Optimized_Access := 'TRUE' }
VERSION : 0.1
// stored: AutoNumber true, IsIECCheckEnabled false, SetENOAutomatically false, UDAEnableTagReadback false
BEGIN

REGION Network 1: Se Bomba 1 Avariar ficam a trabalhar a Bomba 2 e Bomba 3
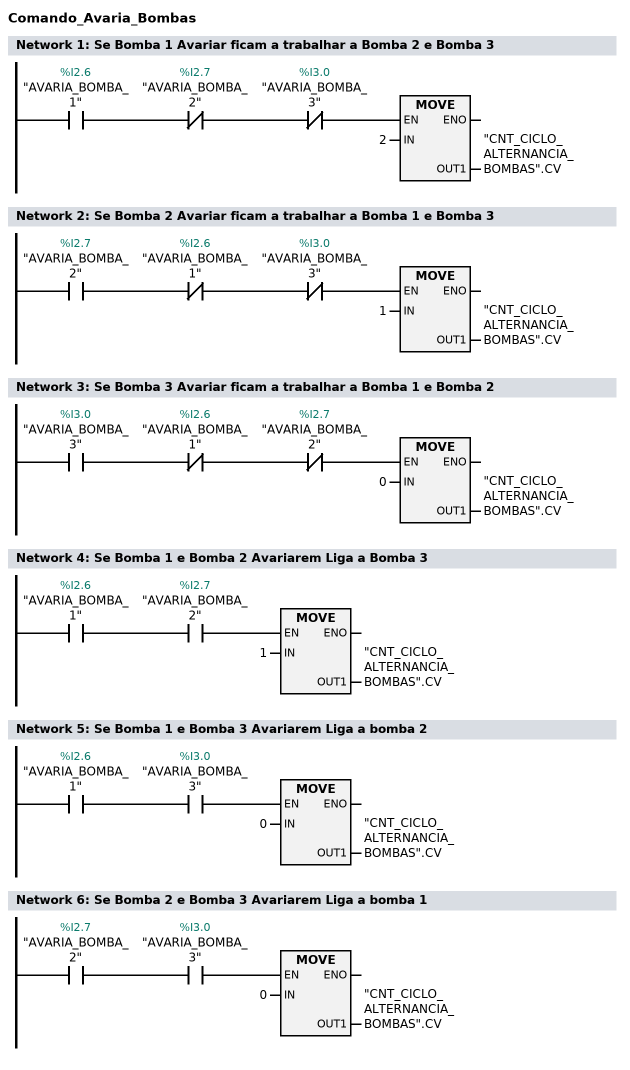
   RUNG wire#powerrail
      Contact( "AVARIA_BOMBA_1" )
      I_Contact( "AVARIA_BOMBA_2" )
      I_Contact( "AVARIA_BOMBA_3" )
      Move(in := 2, out1 => "CNT_CICLO_ALTERNANCIA_BOMBAS".CV)
   END_RUNG
   // the same network as SCL:
   IF "AVARIA_BOMBA_1" AND NOT "AVARIA_BOMBA_2" AND NOT "AVARIA_BOMBA_3" THEN
       "CNT_CICLO_ALTERNANCIA_BOMBAS".CV := 2;
   END_IF;
END_REGION

REGION Network 2: Se Bomba 2 Avariar ficam a trabalhar a Bomba 1 e Bomba 3
   RUNG wire#powerrail
      Contact( "AVARIA_BOMBA_2" )
      I_Contact( "AVARIA_BOMBA_1" )
      I_Contact( "AVARIA_BOMBA_3" )
      Move(in := 1, out1 => "CNT_CICLO_ALTERNANCIA_BOMBAS".CV)
   END_RUNG
   // the same network as SCL:
   IF "AVARIA_BOMBA_2" AND NOT "AVARIA_BOMBA_1" AND NOT "AVARIA_BOMBA_3" THEN
       "CNT_CICLO_ALTERNANCIA_BOMBAS".CV := 1;
   END_IF;
END_REGION

REGION Network 3: Se Bomba 3 Avariar ficam a trabalhar a Bomba 1 e Bomba 2
   RUNG wire#powerrail
      Contact( "AVARIA_BOMBA_3" )
      I_Contact( "AVARIA_BOMBA_1" )
      I_Contact( "AVARIA_BOMBA_2" )
      Move(in := 0, out1 => "CNT_CICLO_ALTERNANCIA_BOMBAS".CV)
   END_RUNG
   // the same network as SCL:
   IF "AVARIA_BOMBA_3" AND NOT "AVARIA_BOMBA_1" AND NOT "AVARIA_BOMBA_2" THEN
       "CNT_CICLO_ALTERNANCIA_BOMBAS".CV := 0;
   END_IF;
END_REGION

REGION Network 4: Se Bomba 1 e Bomba 2 Avariarem Liga a Bomba 3
   RUNG wire#powerrail
      Contact( "AVARIA_BOMBA_1" )
      Contact( "AVARIA_BOMBA_2" )
      Move(in := 1, out1 => "CNT_CICLO_ALTERNANCIA_BOMBAS".CV)
   END_RUNG
   // the same network as SCL:
   IF "AVARIA_BOMBA_1" AND "AVARIA_BOMBA_2" THEN "CNT_CICLO_ALTERNANCIA_BOMBAS".CV := 1; END_IF;
END_REGION

REGION Network 5: Se Bomba 1 e Bomba 3 Avariarem Liga a bomba 2
   RUNG wire#powerrail
      Contact( "AVARIA_BOMBA_1" )
      Contact( "AVARIA_BOMBA_3" )
      Move(in := 0, out1 => "CNT_CICLO_ALTERNANCIA_BOMBAS".CV)
   END_RUNG
   // the same network as SCL:
   IF "AVARIA_BOMBA_1" AND "AVARIA_BOMBA_3" THEN "CNT_CICLO_ALTERNANCIA_BOMBAS".CV := 0; END_IF;
END_REGION

REGION Network 6: Se Bomba 2 e Bomba 3 Avariarem Liga a bomba 1
   RUNG wire#powerrail
      Contact( "AVARIA_BOMBA_2" )
      Contact( "AVARIA_BOMBA_3" )
      Move(in := 0, out1 => "CNT_CICLO_ALTERNANCIA_BOMBAS".CV)
   END_RUNG
   // the same network as SCL:
   IF "AVARIA_BOMBA_2" AND "AVARIA_BOMBA_3" THEN "CNT_CICLO_ALTERNANCIA_BOMBAS".CV := 0; END_IF;
END_REGION
END_FUNCTION

DATA_BLOCK "CNT_CICLO_ALTERNANCIA_BOMBAS"   // DB12
{ S7_Optimized_Access := 'TRUE' }
// stored: AutoNumber true, InstanceOfName IEC_COUNTER, OfSystemLibElement IEC_COUNTER, OfSystemLibVersion 1.0
"IEC_COUNTER"
   // VAR RETAIN
   //    CU : Bool;
   //    CD : Bool;
   //    R : Bool;
   //    LD : Bool;
   //    QU : Bool;
   //    QD : Bool;
   //    PV : Int;
   //    CV : Int;
   // END_VAR
BEGIN
END_DATA_BLOCK

DATA_BLOCK "CNT_FUNC_B1"   // DB14
{ S7_Optimized_Access := 'TRUE' }
// stored: AutoNumber true, InstanceOfName IEC_COUNTER, OfSystemLibElement IEC_COUNTER, OfSystemLibVersion 1.0
"IEC_COUNTER"
   // VAR RETAIN
   //    CU : Bool;
   //    CD : Bool;
   //    R : Bool;
   //    LD : Bool;
   //    QU : Bool;
   //    QD : Bool;
   //    PV : Int;
   //    CV : Int;
   // END_VAR
BEGIN
END_DATA_BLOCK

DATA_BLOCK "CNT_FUNC_B2"   // DB37
{ S7_Optimized_Access := 'TRUE' }
// stored: AutoNumber true, InstanceOfName IEC_COUNTER, OfSystemLibElement IEC_COUNTER, OfSystemLibVersion 1.0
"IEC_COUNTER"
   // VAR RETAIN
   //    CU : Bool;
   //    CD : Bool;
   //    R : Bool;
   //    LD : Bool;
   //    QU : Bool;
   //    QD : Bool;
   //    PV : Int;
   //    CV : Int;
   // END_VAR
BEGIN
END_DATA_BLOCK

DATA_BLOCK "CNT_FUNC_B3"   // DB39
{ S7_Optimized_Access := 'TRUE' }
// stored: AutoNumber true, InstanceOfName IEC_COUNTER, OfSystemLibElement IEC_COUNTER, OfSystemLibVersion 1.0
"IEC_COUNTER"
   // VAR RETAIN
   //    CU : Bool;
   //    CD : Bool;
   //    R : Bool;
   //    LD : Bool;
   //    QU : Bool;
   //    QD : Bool;
   //    PV : Int;
   //    CV : Int;
   // END_VAR
BEGIN
END_DATA_BLOCK

DATA_BLOCK "Hold_Pulse"   // DB41
{ S7_Optimized_Access := 'TRUE' }
// stored: AutoNumber true, InstanceOfName IEC_TIMER, OfSystemLibElement IEC_TIMER, OfSystemLibVersion 1.0
"IEC_TIMER"
   // VAR
   //    PT : Time;
   //    ET { ExternalWritable := 'False'} : Time;
   //    IN : Bool;
   //    Q { ExternalWritable := 'False'} : Bool;
   // END_VAR
BEGIN
END_DATA_BLOCK

DATA_BLOCK "PERÍODO_ALTERNANCIA_BOMBAS"   // DB10
{ S7_Optimized_Access := 'TRUE' }
// stored: AutoNumber true, InstanceOfName IEC_TIMER, OfSystemLibElement IEC_TIMER, OfSystemLibVersion 1.0
"IEC_TIMER"
   // VAR RETAIN
   //    PT : Time;
   //    ET { ExternalWritable := 'False'} : Time;
   //    IN : Bool;
   //    Q { ExternalWritable := 'False'} : Bool;
   // END_VAR
BEGIN
END_DATA_BLOCK

DATA_BLOCK "TEMP_FUNC_B1"   // DB13
{ S7_Optimized_Access := 'TRUE' }
// stored: AutoNumber true, InstanceOfName IEC_TIMER, OfSystemLibElement IEC_TIMER, OfSystemLibVersion 1.0
"IEC_TIMER"
   // VAR
   //    PT : Time;
   //    ET { ExternalWritable := 'False'} : Time;
   //    IN : Bool;
   //    Q { ExternalWritable := 'False'} : Bool;
   // END_VAR
BEGIN
END_DATA_BLOCK

DATA_BLOCK "TEMP_FUNC_B2"   // DB15
{ S7_Optimized_Access := 'TRUE' }
// stored: AutoNumber true, InstanceOfName IEC_TIMER, OfSystemLibElement IEC_TIMER, OfSystemLibVersion 1.0
"IEC_TIMER"
   // VAR
   //    PT : Time;
   //    ET { ExternalWritable := 'False'} : Time;
   //    IN : Bool;
   //    Q { ExternalWritable := 'False'} : Bool;
   // END_VAR
BEGIN
END_DATA_BLOCK

DATA_BLOCK "TEMP_FUNC_B3"   // DB38
{ S7_Optimized_Access := 'TRUE' }
// stored: AutoNumber true, InstanceOfName IEC_TIMER, OfSystemLibElement IEC_TIMER, OfSystemLibVersion 1.0
"IEC_TIMER"
   // VAR
   //    PT : Time;
   //    ET { ExternalWritable := 'False'} : Time;
   //    IN : Bool;
   //    Q { ExternalWritable := 'False'} : Bool;
   // END_VAR
BEGIN
END_DATA_BLOCK

DATA_BLOCK "T_ABERTURA_EV1.1_HMI"   // DB16
{ S7_Optimized_Access := 'TRUE' }
// stored: AutoNumber true, InstanceOfName IEC_TIMER, OfSystemLibElement IEC_TIMER, OfSystemLibVersion 1.0
"IEC_TIMER"
   // VAR
   //    PT : Time;
   //    ET { ExternalWritable := 'False'} : Time;
   //    IN : Bool;
   //    Q { ExternalWritable := 'False'} : Bool;
   // END_VAR
BEGIN
END_DATA_BLOCK

DATA_BLOCK "T_ABERTURA_EV1.2_HMI"   // DB27
{ S7_Optimized_Access := 'TRUE' }
// stored: AutoNumber true, InstanceOfName IEC_TIMER, OfSystemLibElement IEC_TIMER, OfSystemLibVersion 1.0
"IEC_TIMER"
   // VAR
   //    PT : Time;
   //    ET { ExternalWritable := 'False'} : Time;
   //    IN : Bool;
   //    Q { ExternalWritable := 'False'} : Bool;
   // END_VAR
BEGIN
END_DATA_BLOCK

DATA_BLOCK "T_ABERTURA_EV2.1_HMI"   // DB19
{ S7_Optimized_Access := 'TRUE' }
// stored: AutoNumber true, InstanceOfName IEC_TIMER, OfSystemLibElement IEC_TIMER, OfSystemLibVersion 1.0
"IEC_TIMER"
   // VAR
   //    PT : Time;
   //    ET { ExternalWritable := 'False'} : Time;
   //    IN : Bool;
   //    Q { ExternalWritable := 'False'} : Bool;
   // END_VAR
BEGIN
END_DATA_BLOCK

DATA_BLOCK "T_ABERTURA_EV2.2_HMI"   // DB29
{ S7_Optimized_Access := 'TRUE' }
// stored: AutoNumber true, InstanceOfName IEC_TIMER, OfSystemLibElement IEC_TIMER, OfSystemLibVersion 1.0
"IEC_TIMER"
   // VAR
   //    PT : Time;
   //    ET { ExternalWritable := 'False'} : Time;
   //    IN : Bool;
   //    Q { ExternalWritable := 'False'} : Bool;
   // END_VAR
BEGIN
END_DATA_BLOCK

DATA_BLOCK "T_ABERTURA_EV3.1_HMI"   // DB21
{ S7_Optimized_Access := 'TRUE' }
// stored: AutoNumber true, InstanceOfName IEC_TIMER, OfSystemLibElement IEC_TIMER, OfSystemLibVersion 1.0
"IEC_TIMER"
   // VAR
   //    PT : Time;
   //    ET { ExternalWritable := 'False'} : Time;
   //    IN : Bool;
   //    Q { ExternalWritable := 'False'} : Bool;
   // END_VAR
BEGIN
END_DATA_BLOCK

DATA_BLOCK "T_ABERTURA_EV3.2_HMI"   // DB31
{ S7_Optimized_Access := 'TRUE' }
// stored: AutoNumber true, InstanceOfName IEC_TIMER, OfSystemLibElement IEC_TIMER, OfSystemLibVersion 1.0
"IEC_TIMER"
   // VAR
   //    PT : Time;
   //    ET { ExternalWritable := 'False'} : Time;
   //    IN : Bool;
   //    Q { ExternalWritable := 'False'} : Bool;
   // END_VAR
BEGIN
END_DATA_BLOCK

DATA_BLOCK "T_ABERTURA_EV4.1_HMI"   // DB23
{ S7_Optimized_Access := 'TRUE' }
// stored: AutoNumber true, InstanceOfName IEC_TIMER, OfSystemLibElement IEC_TIMER, OfSystemLibVersion 1.0
"IEC_TIMER"
   // VAR
   //    PT : Time;
   //    ET { ExternalWritable := 'False'} : Time;
   //    IN : Bool;
   //    Q { ExternalWritable := 'False'} : Bool;
   // END_VAR
BEGIN
END_DATA_BLOCK

DATA_BLOCK "T_ABERTURA_EV4.2_HMI"   // DB33
{ S7_Optimized_Access := 'TRUE' }
// stored: AutoNumber true, InstanceOfName IEC_TIMER, OfSystemLibElement IEC_TIMER, OfSystemLibVersion 1.0
"IEC_TIMER"
   // VAR
   //    PT : Time;
   //    ET { ExternalWritable := 'False'} : Time;
   //    IN : Bool;
   //    Q { ExternalWritable := 'False'} : Bool;
   // END_VAR
BEGIN
END_DATA_BLOCK

DATA_BLOCK "T_ABERTURA_EV5.1_HMI"   // DB25
{ S7_Optimized_Access := 'TRUE' }
// stored: AutoNumber true, InstanceOfName IEC_TIMER, OfSystemLibElement IEC_TIMER, OfSystemLibVersion 1.0
"IEC_TIMER"
   // VAR
   //    PT : Time;
   //    ET { ExternalWritable := 'False'} : Time;
   //    IN : Bool;
   //    Q { ExternalWritable := 'False'} : Bool;
   // END_VAR
BEGIN
END_DATA_BLOCK

DATA_BLOCK "T_ABERTURA_EV5.2_HMI"   // DB35
{ S7_Optimized_Access := 'TRUE' }
// stored: AutoNumber true, InstanceOfName IEC_TIMER, OfSystemLibElement IEC_TIMER, OfSystemLibVersion 1.0
"IEC_TIMER"
   // VAR
   //    PT : Time;
   //    ET { ExternalWritable := 'False'} : Time;
   //    IN : Bool;
   //    Q { ExternalWritable := 'False'} : Bool;
   // END_VAR
BEGIN
END_DATA_BLOCK

DATA_BLOCK "T_FECHO_EV1.1_HMI"   // DB17
{ S7_Optimized_Access := 'TRUE' }
// stored: AutoNumber true, InstanceOfName IEC_TIMER, OfSystemLibElement IEC_TIMER, OfSystemLibVersion 1.0
"IEC_TIMER"
   // VAR
   //    PT : Time;
   //    ET { ExternalWritable := 'False'} : Time;
   //    IN : Bool;
   //    Q { ExternalWritable := 'False'} : Bool;
   // END_VAR
BEGIN
END_DATA_BLOCK

DATA_BLOCK "T_FECHO_EV1.2_HMI"   // DB28
{ S7_Optimized_Access := 'TRUE' }
// stored: AutoNumber true, InstanceOfName IEC_TIMER, OfSystemLibElement IEC_TIMER, OfSystemLibVersion 1.0
"IEC_TIMER"
   // VAR
   //    PT : Time;
   //    ET { ExternalWritable := 'False'} : Time;
   //    IN : Bool;
   //    Q { ExternalWritable := 'False'} : Bool;
   // END_VAR
BEGIN
END_DATA_BLOCK

DATA_BLOCK "T_FECHO_EV2.1_HMI"   // DB20
{ S7_Optimized_Access := 'TRUE' }
// stored: AutoNumber true, InstanceOfName IEC_TIMER, OfSystemLibElement IEC_TIMER, OfSystemLibVersion 1.0
"IEC_TIMER"
   // VAR
   //    PT : Time;
   //    ET { ExternalWritable := 'False'} : Time;
   //    IN : Bool;
   //    Q { ExternalWritable := 'False'} : Bool;
   // END_VAR
BEGIN
END_DATA_BLOCK

DATA_BLOCK "T_FECHO_EV2.2_HMI"   // DB30
{ S7_Optimized_Access := 'TRUE' }
// stored: AutoNumber true, InstanceOfName IEC_TIMER, OfSystemLibElement IEC_TIMER, OfSystemLibVersion 1.0
"IEC_TIMER"
   // VAR
   //    PT : Time;
   //    ET { ExternalWritable := 'False'} : Time;
   //    IN : Bool;
   //    Q { ExternalWritable := 'False'} : Bool;
   // END_VAR
BEGIN
END_DATA_BLOCK

DATA_BLOCK "T_FECHO_EV3.1_HMI"   // DB22
{ S7_Optimized_Access := 'TRUE' }
// stored: AutoNumber true, InstanceOfName IEC_TIMER, OfSystemLibElement IEC_TIMER, OfSystemLibVersion 1.0
"IEC_TIMER"
   // VAR
   //    PT : Time;
   //    ET { ExternalWritable := 'False'} : Time;
   //    IN : Bool;
   //    Q { ExternalWritable := 'False'} : Bool;
   // END_VAR
BEGIN
END_DATA_BLOCK

DATA_BLOCK "T_FECHO_EV3.2_HMI"   // DB32
{ S7_Optimized_Access := 'TRUE' }
// stored: AutoNumber true, InstanceOfName IEC_TIMER, OfSystemLibElement IEC_TIMER, OfSystemLibVersion 1.0
"IEC_TIMER"
   // VAR
   //    PT : Time;
   //    ET { ExternalWritable := 'False'} : Time;
   //    IN : Bool;
   //    Q { ExternalWritable := 'False'} : Bool;
   // END_VAR
BEGIN
END_DATA_BLOCK

DATA_BLOCK "T_FECHO_EV4.1_HMI"   // DB24
{ S7_Optimized_Access := 'TRUE' }
// stored: AutoNumber true, InstanceOfName IEC_TIMER, OfSystemLibElement IEC_TIMER, OfSystemLibVersion 1.0
"IEC_TIMER"
   // VAR
   //    PT : Time;
   //    ET { ExternalWritable := 'False'} : Time;
   //    IN : Bool;
   //    Q { ExternalWritable := 'False'} : Bool;
   // END_VAR
BEGIN
END_DATA_BLOCK

DATA_BLOCK "T_FECHO_EV4.2_HMI"   // DB34
{ S7_Optimized_Access := 'TRUE' }
// stored: AutoNumber true, InstanceOfName IEC_TIMER, OfSystemLibElement IEC_TIMER, OfSystemLibVersion 1.0
"IEC_TIMER"
   // VAR
   //    PT : Time;
   //    ET { ExternalWritable := 'False'} : Time;
   //    IN : Bool;
   //    Q { ExternalWritable := 'False'} : Bool;
   // END_VAR
BEGIN
END_DATA_BLOCK

DATA_BLOCK "T_FECHO_EV5.1_HMI"   // DB26
{ S7_Optimized_Access := 'TRUE' }
// stored: AutoNumber true, InstanceOfName IEC_TIMER, OfSystemLibElement IEC_TIMER, OfSystemLibVersion 1.0
"IEC_TIMER"
   // VAR
   //    PT : Time;
   //    ET { ExternalWritable := 'False'} : Time;
   //    IN : Bool;
   //    Q { ExternalWritable := 'False'} : Bool;
   // END_VAR
BEGIN
END_DATA_BLOCK

DATA_BLOCK "T_FECHO_EV5.2_HMI"   // DB36
{ S7_Optimized_Access := 'TRUE' }
// stored: AutoNumber true, InstanceOfName IEC_TIMER, OfSystemLibElement IEC_TIMER, OfSystemLibVersion 1.0
"IEC_TIMER"
   // VAR
   //    PT : Time;
   //    ET { ExternalWritable := 'False'} : Time;
   //    IN : Bool;
   //    Q { ExternalWritable := 'False'} : Bool;
   // END_VAR
BEGIN
END_DATA_BLOCK

DATA_BLOCK "T_LAVAGEM"   // DB4
{ S7_Optimized_Access := 'TRUE' }
// stored: AutoNumber true, InstanceOfName IEC_TIMER, OfSystemLibElement IEC_TIMER, OfSystemLibVersion 1.0
"IEC_TIMER"
   // VAR RETAIN
   //    PT : Time;
   //    ET { ExternalWritable := 'False'} : Time;
   //    IN : Bool;
   //    Q { ExternalWritable := 'False'} : Bool;
   // END_VAR
BEGIN
END_DATA_BLOCK

DATA_BLOCK "T_POS_EVS"   // DB3
{ S7_Optimized_Access := 'TRUE' }
// stored: AutoNumber true, InstanceOfName IEC_TIMER, OfSystemLibElement IEC_TIMER, OfSystemLibVersion 1.0
"IEC_TIMER"
   // VAR
   //    PT : Time;
   //    ET { ExternalWritable := 'False'} : Time;
   //    IN : Bool;
   //    Q { ExternalWritable := 'False'} : Bool;
   // END_VAR
BEGIN
END_DATA_BLOCK

DATA_BLOCK "T_PRESS_FILT_1"   // DB8
{ S7_Optimized_Access := 'TRUE' }
// stored: AutoNumber true, InstanceOfName IEC_TIMER, OfSystemLibElement IEC_TIMER, OfSystemLibVersion 1.0
"IEC_TIMER"
   // VAR
   //    PT : Time;
   //    ET { ExternalWritable := 'False'} : Time;
   //    IN : Bool;
   //    Q { ExternalWritable := 'False'} : Bool;
   // END_VAR
BEGIN
END_DATA_BLOCK

DATA_BLOCK "T_PRESS_FILT_2"   // DB9
{ S7_Optimized_Access := 'TRUE' }
// stored: AutoNumber true, InstanceOfName IEC_TIMER, OfSystemLibElement IEC_TIMER, OfSystemLibVersion 1.0
"IEC_TIMER"
   // VAR
   //    PT : Time;
   //    ET { ExternalWritable := 'False'} : Time;
   //    IN : Bool;
   //    Q { ExternalWritable := 'False'} : Bool;
   // END_VAR
BEGIN
END_DATA_BLOCK

DATA_BLOCK "T_RINSE"   // DB5
{ S7_Optimized_Access := 'TRUE' }
// stored: AutoNumber true, InstanceOfName IEC_TIMER, OfSystemLibElement IEC_TIMER, OfSystemLibVersion 1.0
"IEC_TIMER"
   // VAR RETAIN
   //    PT : Time;
   //    ET { ExternalWritable := 'False'} : Time;
   //    IN : Bool;
   //    Q { ExternalWritable := 'False'} : Bool;
   // END_VAR
BEGIN
END_DATA_BLOCK

DATA_BLOCK "T_STOP_BOMBAS"   // DB2
{ S7_Optimized_Access := 'TRUE' }
// stored: AutoNumber true, InstanceOfName IEC_TIMER, OfSystemLibElement IEC_TIMER, OfSystemLibVersion 1.0
"IEC_TIMER"
   // VAR
   //    PT : Time;
   //    ET { ExternalWritable := 'False'} : Time;
   //    IN : Bool;
   //    Q { ExternalWritable := 'False'} : Bool;
   // END_VAR
BEGIN
END_DATA_BLOCK
